// TIA Portal V17 export
// export: Created 2023-12-05T13:40:23.5880688Z, ExportSetting WithDefaults, DisplayName Totally Integrated Automation Portal, DisplayVersion V17, DisplayName TIA Portal Openness, DisplayVersion V17, DisplayName TIA Portal Version Control Interface, DisplayVersion V17, DisplayName SINAMICS Startdrive Advanced, DisplayVersion V17, DisplayName SINAMICS Startdrive G130, G150, S120, S150, SINAMICS MV, S210, DisplayVersion V17, DisplayName SINAMICS Startdrive G110M, G120, G120C, G120D, G120P, G115D, DisplayVersion V17, DisplayName STEP 7 Professional, DisplayVersion V17, DisplayName STEP 7 Safety, DisplayVersion V17, DisplayName WinCC Professional, DisplayVersion V17
FUNCTION "FC511 TimeCounterINT" : Void   // FC511, LAD
TITLE = PRODUCTION TIMERS
{ S7_Optimized_Access := 'FALSE' }
AUTHOR : CER
VERSION : 0.1
// stored: AutoNumber false, IsIECCheckEnabled false, SetENOAutomatically false, UDAEnableTagReadback false
   VAR_INPUT
      START : Bool;   // ENABLE TIMER
      STOP : Bool;   // RESET TIMER
      PULSE : Bool;   // PULSE SIGNAL
      DECLARED_TIME : Int;   // Max time
   END_VAR
   VAR_IN_OUT
      ACTUAL_TIME : Int;   // Actual time
      FP_Bit : Bool;   // FP Start
      TIME_REACHED : Bool;   // Max time reached
   END_VAR
BEGIN

NETWORK
TITLE = Max time reached
      O     #STOP;
      O     #TIME_REACHED;
      JC    rset;

      A     #START;
      AN    #TIME_REACHED;
      A     #PULSE;
      FP    #FP_Bit;
      JC    time;
      BEU;

time: L     #ACTUAL_TIME;
      L     1;
      +I;
      T     #ACTUAL_TIME;
      L     #ACTUAL_TIME;
      L     #DECLARED_TIME;
      >=I;
      S     #TIME_REACHED;
      BEU;

rset: L     0;
      T     #ACTUAL_TIME;
      BEU;



END_FUNCTION
